FUNCTION_BLOCK FB_LinearMovementWithFeedbackTest EXTENDS FB_TestSuite
VAR_INPUT
END_VAR
VAR_OUTPUT
END_VAR
VAR
END_VAR

Movement_stops_when_position_is_reached();
Movement_executes_when_triggered();
Output_is_still_active_when_position_has_been_reached_but_holdPos_has_been_set();
No_Movement_When_Direction_Is_Locked();

METHOD Movement_executes_when_triggered : BOOL
VAR_INPUT
END_VAR
VAR
	sut: FB_LinearMovementWithFeedback;
	result : BOOL := TRUE;
END_VAR
TEST('Movement executes when triggered');

sut(
	ToPosition:= TRUE,
	Feedback:= FALSE,
	Lock:= FALSE,
	HoldOutput:= FALSE);
	
AssertEquals(result, sut.Actor, 'Movement does not start');

TEST_FINISHED();
END_METHOD

METHOD Movement_stops_when_position_is_reached : BOOL
VAR_INPUT
END_VAR
VAR_INST
	sut: FB_LinearMovementWithFeedback;
	result : BOOL := FALSE;
END_VAR
TEST('Movement stops when position is reached');

sut(
	ToPosition:= TRUE,
	Feedback:= True,
	Lock:= FALSE,
	HoldOutput:= FALSE);
	
AssertEquals(result, sut.Actor, 'Movement even if not enabled');

TEST_FINISHED();
END_METHOD

METHOD No_Movement_When_Direction_Is_Locked : BOOL
VAR_INPUT
END_VAR
VAR
	sut: FB_LinearMovementWithFeedback;
	result : BOOL := FALSE;
END_VAR
TEST('Output should remain set when position is reached but Hold is set');

sut(
	ToPosition:= TRUE,
	Feedback:= FALSE,
	Lock:= TRUE,
	HoldOutput:= FALSE);
	
AssertEquals(result, sut.Actor, 'Target reached but output not hold.');

TEST_FINISHED();
END_METHOD

METHOD Output_is_still_active_when_position_has_been_reached_but_holdPos_has_been_set : BOOL
VAR_INPUT
END_VAR
VAR
	sut: FB_LinearMovementWithFeedback;
	result : BOOL := TRUE;
END_VAR
TEST('Output remains set when position has been reached when setting hold pos is true');

sut(
	ToPosition:= TRUE,
	Feedback:= True,
	Lock:= FALSE,
	HoldOutput:= TRUE);
	
AssertEquals(result, sut.Actor, '');

TEST_FINISHED();
END_METHOD

END_FUNCTION_BLOCK

(* stored: Version 1.1.0.1, ProductVersion 3.1.4024.11
   POU FB_LinearMovementWithFeedbackTest: Id {a4f63ed1-56b1-4e6a-95e3-66dd048248da}, SpecialFunc None
   Method Movement_executes_when_triggered: Id {665bda91-0ea2-4739-b488-2974f55cf3db}
   Method Movement_stops_when_position_is_reached: Id {c6fe306a-d96b-44dd-8f7e-92ce75c0cfb9}
   Method No_Movement_When_Direction_Is_Locked: Id {c91f3a13-b3c7-4c01-8905-9da15cf0d01c}
   Method Output_is_still_active_when_position_has_been_reached_but_holdPos_has_been_set: Id {8b1a8142-d64c-4aa8-b645-31f96c78c98e} *)
